PROGRAM get_images
VAR
	start_head: BOOL;
	start_nut : BOOL;
	vi_get_img_cabezal_dere : BOOL;
	vi_get_img_nut : BOOL;
	head_ok : BOOL;
	nut_ok : BOOL;
END_VAR

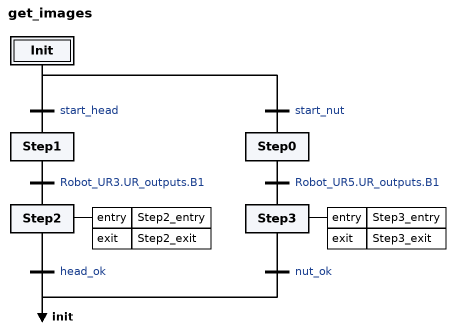
INITIAL_STEP Init:
END_STEP
TRANSITION FROM Init TO Step1
    := start_head;
END_TRANSITION
STEP Step1:
END_STEP
TRANSITION FROM Step1 TO Step2
    := Robot_UR3.UR_outputs.B1;
END_TRANSITION
STEP Step2:
    Step2_entry(P1);  // entry action
    Step2_exit(P0);  // exit action
END_STEP
TRANSITION FROM Step2 TO init
    := head_ok;
END_TRANSITION
TRANSITION FROM Init TO Step0
    := start_nut;
END_TRANSITION
STEP Step0:
END_STEP
TRANSITION FROM Step0 TO Step3
    := Robot_UR5.UR_outputs.B1;
END_TRANSITION
STEP Step3:
    Step3_entry(P1);  // entry action
    Step3_exit(P0);  // exit action
END_STEP
TRANSITION FROM Step3 TO init
    := nut_ok;
END_TRANSITION

ACTION Step2_entry:
vi_get_img_cabezal_dere := TRUE;
Robot_UR3.UR_inputs.Bits.B1 := False;
END_ACTION

ACTION Step2_exit:
vi_get_img_cabezal_dere := FALSE;
Robot_UR3.UR_inputs.Bits.B1 := TRUE;
head_ok := False;
END_ACTION

ACTION Step3_entry:
vi_get_img_nut := TRUE;
Robot_UR5.UR_inputs.Bits.B1 := False;
END_ACTION

ACTION Step3_exit:
vi_get_img_nut := FALSE;
Robot_UR5.UR_inputs.Bits.B1 := TRUE;
nut_ok := False;
END_ACTION

END_PROGRAM

(* stored: Version 1.1.0.1, ProductVersion 3.1.4024.4
   POU get_images: Id {52582e99-c789-46de-a81d-3733b141ed7d}, SpecialFunc None
   Action Step2_entry: Id {3e95e87f-e532-42fa-b7cf-c206a94d0d10}
   Action Step2_exit: Id {e565ee66-68a9-4612-a693-858af2dda7e8}
   Action Step3_entry: Id {4c9b0646-b72f-472b-9d6e-f28482a9fde3}
   Action Step3_exit: Id {9f3625b9-9377-40f9-87be-58253f8253d4} *)
